
FUNCTION CB_add_time : TIME


TITLE = ' Adding two duration '
VERSION : '1.0'
AUTHOR  : CB
NAME    : add_time
FAMILY  : TNI

VAR_INPUT
    IN0 : TIME;
    IN1 : TIME;
END_VAR

BEGIN
    CB_add_time := IN0 + IN1;
END_FUNCTION
